SUBAPPLICATION Uebung_007d2_AX (* Blinker mit E_CYCLE, FB_AR_RANDOM, AR_GT und AX_D_FF_TMIN *)
  (* Standard: 61499-2; Description: Copyright (c) 2023 Meisterschulen am Ostbahnhof This program and the accompanying materials are made available under the terms of the Eclipse Public License 2.0 which is available at https://www.eclipse.org/legal/epl-2.0/ SPDX-License-Identifier: EPL-2.0 *)
  (* Version 1.0, 2023-10-23, Franz Höpfinger, Meisterschulen am Ostbahnhof, initial API and implementation and/or initial documentation *)
  PACKAGE Uebungen;
  IMPORT logiBUS::io::DQ::logiBUS_DO::Output_Q1;
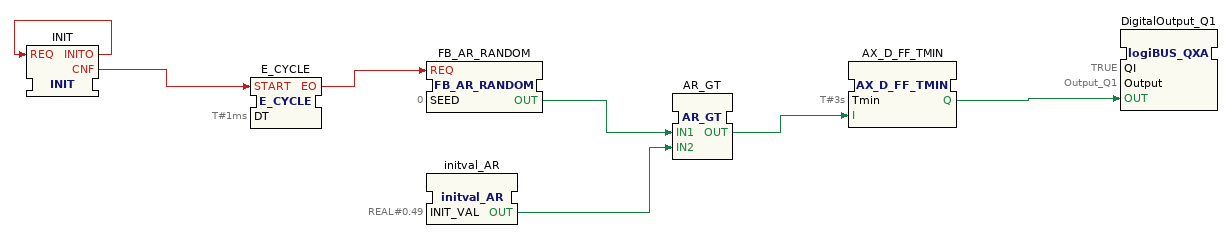
  FBS
    DigitalOutput_Q1 : logiBUS::io::DQ::logiBUS_QXA(QI := TRUE, Output := Output_Q1);
    E_CYCLE : iec61499::events::E_CYCLE(DT := T#1ms);
    FB_AR_RANDOM : adapter::utils::FB_AR_RANDOM(SEED := 0);
    initval_AR : adapter::types::unidirectional::AR::initval::initval_AR(INIT_VAL := REAL#0.49);
    AR_GT : adapter::iec61131::comparison::AR_GT;
    AX_D_FF_TMIN : adapter::events::unidirectional::AX_D_FF_TMIN(Tmin := T#3s);
    INIT : iec61131::booleanOperators::INIT;
  END_FBS
  EVENT_CONNECTIONS
    INIT.INITO TO INIT.REQ;
    INIT.CNF TO E_CYCLE.START;
    E_CYCLE.EO TO FB_AR_RANDOM.REQ;
  END_CONNECTIONS
  ADAPTER_CONNECTIONS
    FB_AR_RANDOM.OUT TO AR_GT.IN1;
    initval_AR.OUT TO AR_GT.IN2;
    AR_GT.OUT TO AX_D_FF_TMIN.I;
    AX_D_FF_TMIN.Q TO DigitalOutput_Q1.OUT;
  END_CONNECTIONS
END_SUBAPPLICATION
